INTERFACE ITF_Group3_HMI_Connector EXTENDS
	ITF_BaseGroupElement_HMI_Connector, ITF_Group3_HMI_Connector_View, ITF_Group3_HMI_Connector_Command

END_INTERFACE

(* stored: Version 1.1.0.1
   Itf ITF_Group3_HMI_Connector: Id {d3cf72ea-bd21-02c9-1e98-e6b7b583a0a5} *)
